FUNCTION F_ConfigPosition



F_ConfigPosition_001();

F_ConfigPosition_002();

END_FUNCTION

(* stored: Version 1.1.0.1, ProductVersion 3.1.4024.9
   POU F_ConfigPosition: Id {d1db5a52-a09a-483f-92a4-d00863491a06}, SpecialFunc None *)
